TYPE Es_CoordenadasCaballeteLadoB :
STRUCT
	CoordenadaFinale_X 							: LREAL ;
	CoordenadaFinale_Y 							: LREAL ;
	CoordenadaFinale_Z 							: LREAL ;
	CoordenadaFinale_J 							: LREAL ;
END_STRUCT
END_TYPE

(* stored: Version 1.1.0.1, ProductVersion 3.1.4024.11
   DUT Es_CoordenadasCaballeteLadoB: Id {ddcf4027-dd82-4f8e-a22a-47bdac34eb2a} *)
